KUKA KRL program: Mes_Loop_Sps.sub

&ACCESS RVO
&COMMENT USER specified PLC program
DEF Mes_Loop_Sps( )



; Please adjust Parameters of SUBMIT_CYCLE () call
; First Parameter SPS_TIME: >= 1 determines duration of one run of loop/endloop in ms
; Second Parameter SPS_PRIO: possible values: #PRIO_NORMAL, #PRIO_HIGH, #PRIO_HIGHEST
SUBMIT_CYCLE (5, #PRIO_HIGHEST)


Mes_InFo_Int()
loop
Mes_InFo_Main()
SUBMIT_CYCLE (5, #PRIO_HIGHEST)
WAIT SEC 0
endloop


END
